// Mitsubishi GX Works2 project: Semáforo com bugs_30.09   PLC: Q03UDV

PROGRAM MAIN
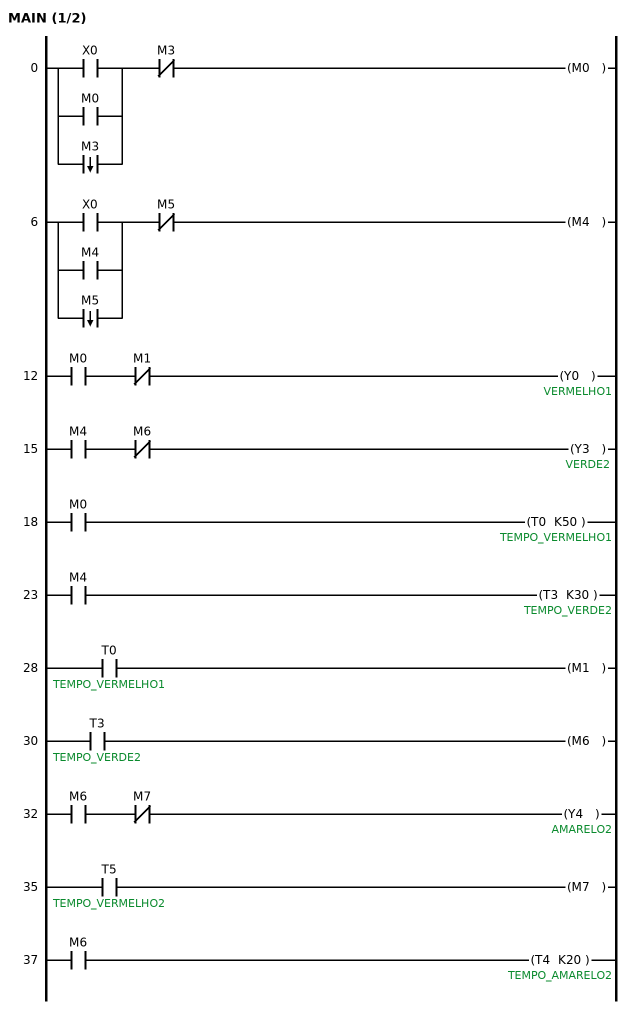
0     LD      X0
      OR      M0
      ORF     M3
      ANI     M3
      OUT     M0
6     LD      X0
      OR      M4
      ORF     M5
      ANI     M5
      OUT     M4
12    LD      M0
      ANI     M1
      OUT     Y0  ; VERMELHO1
15    LD      M4
      ANI     M6
      OUT     Y3  ; VERDE2
18    LD      M0
      OUT     T0 K50  ; TEMPO_VERMELHO1
23    LD      M4
      OUT     T3 K30  ; TEMPO_VERDE2
28    LD      T0  ; TEMPO_VERMELHO1
      OUT     M1
30    LD      T3  ; TEMPO_VERDE2
      OUT     M6
32    LD      M6
      ANI     M7
      OUT     Y4  ; AMARELO2
35    LD      T5  ; TEMPO_VERMELHO2
      OUT     M7
37    LD      M6
      OUT     T4 K20  ; TEMPO_AMARELO2
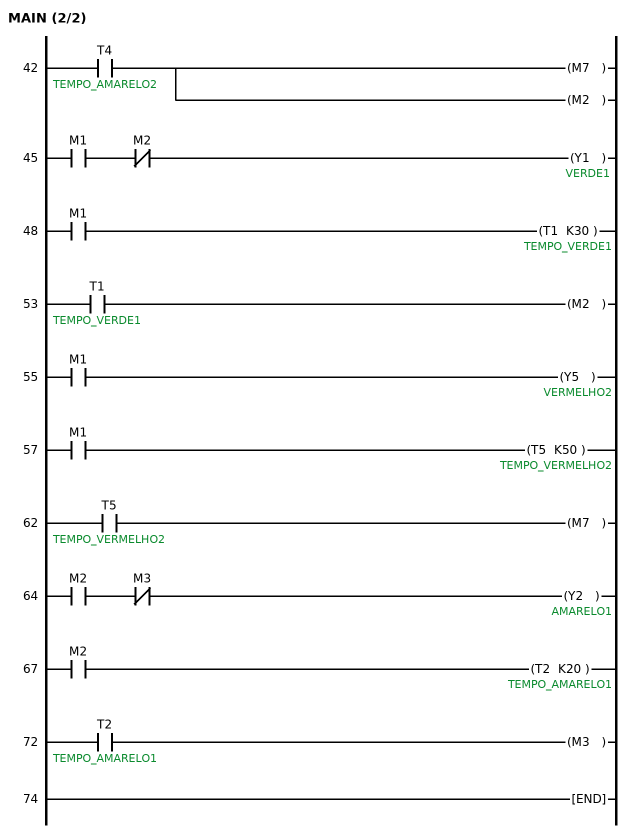
42    LD      T4  ; TEMPO_AMARELO2
      OUT     M7
      OUT     M2
45    LD      M1
      ANI     M2
      OUT     Y1  ; VERDE1
48    LD      M1
      OUT     T1 K30  ; TEMPO_VERDE1
53    LD      T1  ; TEMPO_VERDE1
      OUT     M2
55    LD      M1
      OUT     Y5  ; VERMELHO2
57    LD      M1
      OUT     T5 K50  ; TEMPO_VERMELHO2
62    LD      T5  ; TEMPO_VERMELHO2
      OUT     M7
64    LD      M2
      ANI     M3
      OUT     Y2  ; AMARELO1
67    LD      M2
      OUT     T2 K20  ; TEMPO_AMARELO1
72    LD      T2  ; TEMPO_AMARELO1
      OUT     M3
74    END
END_PROGRAM
